// TIA Portal V20 export
DATA_BLOCK "DB_AnalogInputDataHMI"   // DB1303
TITLE = TEMPERATURE SETTINGS
{ S7_Optimized_Access := 'FALSE'; DB_Accessible_From_OPC_UA := 'FALSE' }
AUTHOR : SAN
// stored: AutoNumber false, DBAccessibleFromOPCUA false, DBAccessibleFromWebserver false
   VAR RETAIN
      Laser_Power_Meter : "AnalogInDataHMI_DT";
      Axis_B_Clamping_Part : "AnalogInDataHMI_DT";
      Laser_Air_Pressure_Process : "AnalogInDataHMI_DT";
      Inlet_Air_Pressure : "AnalogInDataHMI_DT";
      Ambiant_Temperature : "AnalogInDataHMI_DT";
      Machine_Temperature : "AnalogInDataHMI_DT";
      Cold_Water_Temperature_Input : "AnalogInDataHMI_DT";
      Cold_Water_Temperature_Output : "AnalogInDataHMI_DT";
      X_Axis_Temperature_PT1000 { S7_SetPoint := 'True'} : "AnalogInDataHMI_DT";
      Y_Axis_Temperature_PT1000 : "AnalogInDataHMI_DT";
      X_Axis_Temperature_PTC : "AnalogInDataHMI_DT";
      Y_Axis_Temperature_PTC : "AnalogInDataHMI_DT";
      Nozzle_Overpressure : "AnalogInDataHMI_DT";
      Optical_Path_Overpressure : "AnalogInDataHMI_DT";
      Laser_Head_Overpressure : "AnalogInDataHMI_DT";
      ZL_Axis_Overpressure : "AnalogInDataHMI_DT";
      XY_Axis_Overpressure : "AnalogInDataHMI_DT";
      Left_Aspiration : "AnalogInDataHMI_DT";
      Right_Aspiration : "AnalogInDataHMI_DT";
      Free_IW458 : "AnalogInDataHMI_DT";
      Clim_Temperature : "AnalogInDataHMI_DT";
      Free_IW482 : "AnalogInDataHMI_DT";
      Free_IW484 : "AnalogInDataHMI_DT";
      Free_IW486 : "AnalogInDataHMI_DT";
      Sensor_Controller_Station1 : "AnalogInDataHMI_DT";
      Cabinet_Temperature : "AnalogInDataHMI_DT";
      Free_IW464 : "AnalogInDataHMI_DT";
      Free_IW466 : "AnalogInDataHMI_DT";
   END_VAR
BEGIN
   Laser_Power_Meter.ID_Measure := 701;
   Axis_B_Clamping_Part.ID_Measure := 810;
   Laser_Air_Pressure_Process.ID_Measure := 511;
   Laser_Air_Pressure_Process.TargetValue := 2.0;
   Laser_Air_Pressure_Process.ThresholdAlarmMin := -0.2;
   Laser_Air_Pressure_Process.ThresholdWarningMin := -0.15;
   Laser_Air_Pressure_Process.ThresholdWarningMax := 0.15;
   Laser_Air_Pressure_Process.ThresholdAlarmMax := 0.2;
   Laser_Air_Pressure_Process.StartTime := T#5s;
   Inlet_Air_Pressure.ID_Measure := 501;
   Inlet_Air_Pressure.TargetValue := 6.0;
   Inlet_Air_Pressure.ThresholdAlarmMin := -0.5;
   Inlet_Air_Pressure.ThresholdWarningMin := -0.4;
   Inlet_Air_Pressure.ThresholdWarningMax := 0.4;
   Inlet_Air_Pressure.ThresholdAlarmMax := 0.5;
   Inlet_Air_Pressure.StartTime := T#5s;
   Ambiant_Temperature.ID_Measure := 201;
   Ambiant_Temperature.TargetValue := 25.0;
   Ambiant_Temperature.ThresholdAlarmMin := -5.0;
   Ambiant_Temperature.ThresholdWarningMin := -3.0;
   Ambiant_Temperature.ThresholdWarningMax := 3.0;
   Ambiant_Temperature.ThresholdAlarmMax := 5.0;
   Machine_Temperature.ID_Measure := 202;
   Machine_Temperature.TargetValue := 25.0;
   Machine_Temperature.ThresholdAlarmMin := -5.0;
   Machine_Temperature.ThresholdWarningMin := -3.0;
   Machine_Temperature.ThresholdWarningMax := 3.0;
   Machine_Temperature.ThresholdAlarmMax := 5.0;
   Cold_Water_Temperature_Input.ID_Measure := 301;
   Cold_Water_Temperature_Input.TargetValue := 23.0;
   Cold_Water_Temperature_Input.ThresholdAlarmMin := -3.0;
   Cold_Water_Temperature_Input.ThresholdWarningMin := -2.0;
   Cold_Water_Temperature_Input.ThresholdWarningMax := 2.0;
   Cold_Water_Temperature_Input.ThresholdAlarmMax := 3.0;
   Cold_Water_Temperature_Output.ID_Measure := 302;
   Cold_Water_Temperature_Output.TargetValue := 24.0;
   Cold_Water_Temperature_Output.ThresholdAlarmMin := -3.0;
   Cold_Water_Temperature_Output.ThresholdWarningMin := -2.0;
   Cold_Water_Temperature_Output.ThresholdWarningMax := 2.0;
   Cold_Water_Temperature_Output.ThresholdAlarmMax := 3.0;
   X_Axis_Temperature_PT1000.ID_Measure := 110;
   X_Axis_Temperature_PT1000.TargetValue := 25.0;
   X_Axis_Temperature_PT1000.ThresholdAlarmMin := -5.0;
   X_Axis_Temperature_PT1000.ThresholdWarningMin := -3.0;
   X_Axis_Temperature_PT1000.ThresholdWarningMax := 3.0;
   X_Axis_Temperature_PT1000.ThresholdAlarmMax := 5.0;
   X_Axis_Temperature_PT1000.AxFactor := 1.0;
   X_Axis_Temperature_PT1000.StartTime := T#45S;
   Y_Axis_Temperature_PT1000.ID_Measure := 120;
   Y_Axis_Temperature_PT1000.TargetValue := 25.0;
   Y_Axis_Temperature_PT1000.ThresholdAlarmMin := -5.0;
   Y_Axis_Temperature_PT1000.ThresholdWarningMin := -3.0;
   Y_Axis_Temperature_PT1000.ThresholdWarningMax := 3.0;
   Y_Axis_Temperature_PT1000.ThresholdAlarmMax := 5.0;
   X_Axis_Temperature_PTC.ID_Measure := 116;
   Y_Axis_Temperature_PTC.ID_Measure := 126;
   Nozzle_Overpressure.ID_Measure := 512;
   Nozzle_Overpressure.TargetValue := 2.0;
   Nozzle_Overpressure.ThresholdAlarmMin := -0.2;
   Nozzle_Overpressure.ThresholdWarningMin := -0.15;
   Nozzle_Overpressure.ThresholdWarningMax := 0.15;
   Nozzle_Overpressure.ThresholdAlarmMax := 0.2;
   Nozzle_Overpressure.StartTime := T#5s;
   Optical_Path_Overpressure.ID_Measure := 513;
   Optical_Path_Overpressure.TargetValue := 0.4;
   Optical_Path_Overpressure.ThresholdAlarmMin := -0.2;
   Optical_Path_Overpressure.ThresholdWarningMin := -0.19;
   Optical_Path_Overpressure.ThresholdWarningMax := 0.19;
   Optical_Path_Overpressure.ThresholdAlarmMax := 0.2;
   Optical_Path_Overpressure.StartTime := T#5s;
   Laser_Head_Overpressure.ID_Measure := 514;
   Laser_Head_Overpressure.TargetValue := 1.4;
   Laser_Head_Overpressure.ThresholdAlarmMin := -0.15;
   Laser_Head_Overpressure.ThresholdWarningMin := -0.1;
   Laser_Head_Overpressure.ThresholdWarningMax := 0.1;
   Laser_Head_Overpressure.ThresholdAlarmMax := 0.15;
   Laser_Head_Overpressure.StartTime := T#5s;
   ZL_Axis_Overpressure.ID_Measure := 520;
   ZL_Axis_Overpressure.TargetValue := 0.85;
   ZL_Axis_Overpressure.ThresholdAlarmMin := -0.2;
   ZL_Axis_Overpressure.ThresholdWarningMin := -0.15;
   ZL_Axis_Overpressure.ThresholdWarningMax := 0.15;
   ZL_Axis_Overpressure.ThresholdAlarmMax := 0.2;
   ZL_Axis_Overpressure.StartTime := T#5s;
   XY_Axis_Overpressure.ID_Measure := 530;
   XY_Axis_Overpressure.TargetValue := 0.85;
   XY_Axis_Overpressure.ThresholdAlarmMin := -0.2;
   XY_Axis_Overpressure.ThresholdWarningMin := -0.15;
   XY_Axis_Overpressure.ThresholdWarningMax := 0.15;
   XY_Axis_Overpressure.ThresholdAlarmMax := 0.2;
   XY_Axis_Overpressure.StartTime := T#5s;
   Left_Aspiration.ID_Measure := 401;
   Left_Aspiration.CurrentValue := 1.4774;
   Left_Aspiration.TargetValue := 1900.0;
   Left_Aspiration.ThresholdAlarmMin := -1000.0;
   Left_Aspiration.ThresholdWarningMin := -500.0;
   Left_Aspiration.ThresholdWarningMax := 500.0;
   Left_Aspiration.ThresholdAlarmMax := 1000.0;
   Left_Aspiration.StartTime := T#120s;
   Right_Aspiration.ID_Measure := 402;
   Right_Aspiration.CurrentValue := 1.4774;
   Right_Aspiration.TargetValue := 1900.0;
   Right_Aspiration.ThresholdAlarmMin := -1000.0;
   Right_Aspiration.ThresholdWarningMin := -500.0;
   Right_Aspiration.ThresholdWarningMax := 500.0;
   Right_Aspiration.ThresholdAlarmMax := 1000.0;
   Right_Aspiration.StartTime := T#120s;
   Free_IW458.ID_Measure := 999;
   Clim_Temperature.ID_Measure := 204;
   Free_IW482.ID_Measure := 999;
   Free_IW484.ID_Measure := 999;
   Free_IW486.ID_Measure := 999;
   Sensor_Controller_Station1.ID_Measure := 711;
   Cabinet_Temperature.ID_Measure := 203;
   Free_IW464.ID_Measure := 999;
   Free_IW466.ID_Measure := 999;
END_DATA_BLOCK
